FUNCTION_BLOCK FT_PT1 (* Low Pass Filter (PT1) *)
  (* Standard: 61499-1; Description: FT_PT1 is an low pass filter with a programmable time T and faktor K. *)
  (* Version 1.0, 2025-12-21, Franz Höpfinger, initial API and implementation and/or initial documentation *)
  PACKAGE OSCAT::Basic::POUs::Engineering::Control;
  IMPORT OSCAT::Basic::POUs::Engineering::measurements::T_PLC_US;
  IMPORT OSCAT::Basic::POUs::conversion::TIME_TO_REAL;
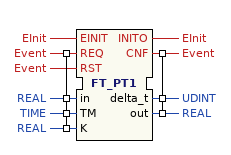
  EVENT_INPUT
    EINIT : EInit; (* Init Request *)
    REQ WITH in, TM, K; (* Normal Execution Request *)
    RST; (* Reset *)
  END_EVENT
  EVENT_OUTPUT
    INITO : EInit; (* Init Confirmation *)
    CNF WITH delta_t, out; (* Execution Confirmation *)
  END_EVENT
  VAR_INPUT
    in : REAL; (* Input Signal *)
    TM : TIME; (* Filter Time Constant *)
    K : REAL := 1.0; (* Gain Factor *)
  END_VAR
  VAR_OUTPUT
    delta_t : UDINT; (* Delta T since last call. *)
    out : REAL; (* Output Signal *)
  END_VAR
  VAR
    last : UDINT; (* Last execution time *)
    tx : UDINT; (* Current execution time *)
    init : BOOL; (* Initialization flag *)
  END_VAR
  EC_STATES
    EINIT : EINIT -> INITO; (* Initialization *)
    REQ : REQ -> CNF; (* Normal Operation *)
    RST : RST -> CNF;
  END_STATES
  ALGORITHM EINIT IN ST:
(* Reset logic *)
init := FALSE;
out := 0.0;
last := UDINT#0;
  END_ALGORITHM
  ALGORITHM RST IN ST:
init := TRUE;
out := K * in;
  END_ALGORITHM
  ALGORITHM REQ IN ST:
(* Read system time *)
tx := T_PLC_US();

(* Startup initialization or T=0 *)
IF NOT init OR TM = T#0s THEN
	this.RST();
ELSE
	(* Calculate time delta since last call *)
	delta_t := (tx - last);

		(* PT1 Formula: out = out + (target - out) * (dt / T) *)
	IF TIME_TO_REAL(TM) > 0.0 THEN
		out := out + (in * K - out) * UDINT_TO_REAL(delta_t) / TIME_TO_REAL(TM);
	END_IF;

		(* Avoid denormalized numbers / underrun *)
	IF ABS(out) < 1.0E-20 THEN
		out := 0.0;
	END_IF;
END_IF;

(* Save time for next cycle *)
last := tx;
  END_ALGORITHM
END_FUNCTION_BLOCK
